(* LS Electric XG5000 project: LM1000_first_NC_program *)
(* PLC LSPLC *)
(* module base 0 slot 0: Input/Output Module:XMC-DN24 (DC 24V Input 8Points/TR output 16Points) *)
(* module base 0 slot 1: Internal Analog Input/Output:XMF-AH04E (A/D voltage/current 2 channels, D/A voltage 2 channels) *)
(* task Periodic Task: Kind=2 *)
(* task Initialization Task: Kind=1 *)
(* task NC Program: Kind=6 *)
VAR_GLOBAL
    NC_Ch1 : UINT := 1;
END_VAR

PROGRAM LDprogram (* task: Scan Program *)
VAR
    LS_CONNECT1 : LS_CONNECT;
    LS_DISCONNECT1 : LS_DISCONNECT;
    MC_HOMEALL1 : MC_HOMEALL;
    MC_POWERALL1 : MC_POWERALL;
    NC_CYCLESTART1 : NC_CYCLESTART;
    NC_LOADPROGRAM1 : NC_LOADPROGRAM;
    NC_RESET1 : NC_RESET;
    xConnect : BOOL;
    xHoming : BOOL;
    xLoadNCProgram : BOOL;
    xResetNCChannel : BOOL;
    xStartCycle : BOOL;
END_VAR
VAR_EXTERNAL
    NC_Ch1 : UINT;
END_VAR
VAR
    _e1 : F_TRIG;
END_VAR

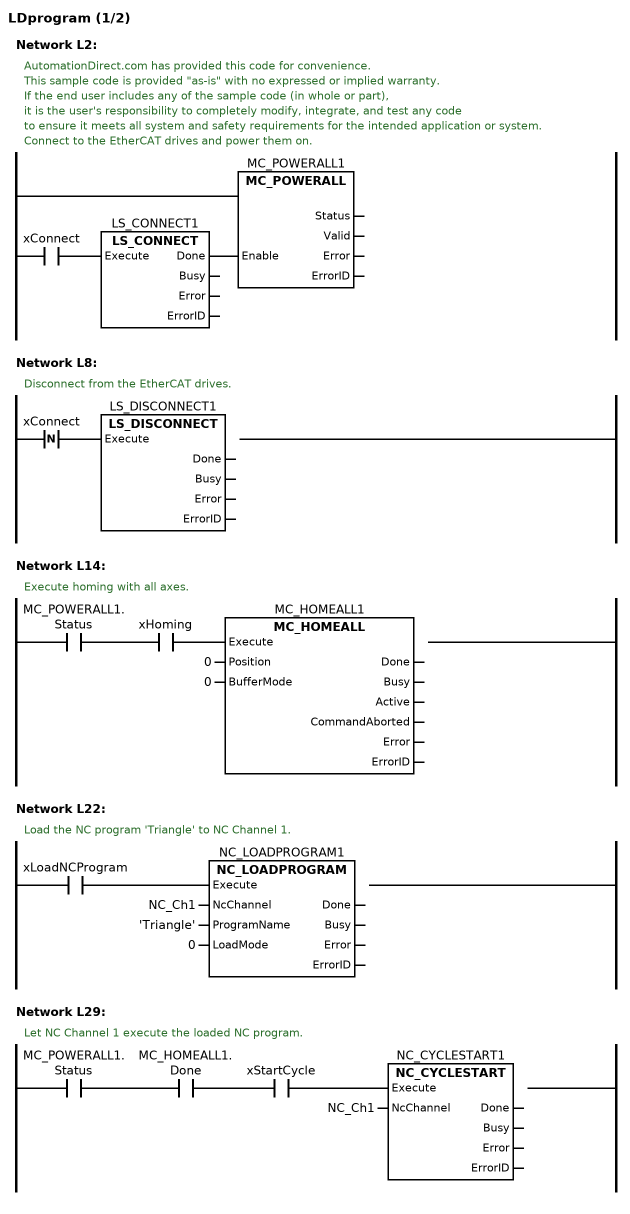
(* AutomationDirect.com has provided this code for convenience. / This sample code is provided "as-is" with no expressed or implied warranty. / If the end user includes any of the sample code (in whole or part), / it is the user's responsibility to completely modify, integrate, and test any code / to ensure it meets all system and safety requirements for the intended application or system. *)
(* Connect to the EtherCAT drives and power them on. *)
(* Rung L2 *)
LS_CONNECT1(Execute := xConnect);
MC_POWERALL1(Enable := LS_CONNECT1.Done);
(* Disconnect from the EtherCAT drives. *)
(* Rung L8 *)
_e1(CLK := xConnect);
LS_DISCONNECT1(Execute := _e1.Q);
(* Execute homing with all axes. *)
(* Rung L14 *)
MC_HOMEALL1(Execute := MC_POWERALL1.Status AND xHoming, Position := 0, BufferMode := 0);
(* Load the NC program 'Triangle' to NC Channel 1. *)
(* Rung L22 *)
NC_LOADPROGRAM1(Execute := xLoadNCProgram, NcChannel := NC_Ch1, ProgramName := 'Triangle', LoadMode := 0);
(* Let NC Channel 1 execute the loaded NC program. *)
(* Rung L29 *)
NC_CYCLESTART1(Execute := MC_POWERALL1.Status AND MC_HOMEALL1.Done AND xStartCycle, NcChannel := NC_Ch1);

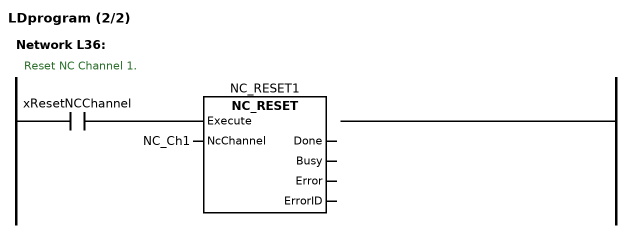
(* Reset NC Channel 1. *)
(* Rung L36 *)
NC_RESET1(Execute := xResetNCChannel, NcChannel := NC_Ch1);
END_PROGRAM

PROGRAM STprogram (* task: Scan Program *)
VAR
    F_TRIG1 : F_TRIG;
    LS_CONNECT1 : LS_CONNECT;
    LS_DISCONNECT1 : LS_DISCONNECT;
    MC_HOMEALL1 : MC_HOMEALL;
    MC_POWERALL1 : MC_POWERALL;
    NC_CYCLESTART1 : NC_CYCLESTART;
    NC_LOADPROGRAM1 : NC_LOADPROGRAM;
    NC_RESET1 : NC_RESET;
    xConnect : BOOL;
    xHoming : BOOL;
    xLoadNCProgram : BOOL;
    xRestNCChannel : BOOL;
    xStartCycle : BOOL;
END_VAR
VAR_EXTERNAL
    NC_Ch1 : UINT;
END_VAR
// AutomationDirect.com has provided this code for convenience. 
// This sample code is provided "as-is" with no expressed or implied warranty. 
// If the end user includes any of the sample code (in whole or part), 
// it is the user's responsibility to completely modify, integrate, and test any code 
// to ensure it meets all system and safety requirements for the intended application or system.


// Connect to the EtherCAT drives and power them on.
LS_CONNECT1(Execute:=xConnect, ErrorID=>LS_CONNECT1.ErrorID);
MC_POWERALL1(Enable:=LS_CONNECT1.Done, ErrorID=>MC_POWERALL1.ErrorID);

// Disconnect from the EtherCAT drives.
F_TRIG1(CLK:=xConnect);
LS_DISCONNECT1(Execute:=F_TRIG1.Q, ErrorID=>LS_DISCONNECT1.ErrorID);

// Execute homing with all axes.
MC_HOMEALL1(Execute:=(MC_POWERALL1.Status AND xHoming), Position:=0, BufferMode:=0, ErrorID=>MC_HOMEALL1.ErrorID);

// Load the NC program 'Triangle' to NC Channel 1.
NC_LOADPROGRAM1(Execute:=xLoadNCProgram, NcChannel:=NC_Ch1, ProgramName:='Triangle', LoadMode:=0, ErrorID=>NC_LOADPROGRAM1.ErrorID);

// Let NC Channel 1 execute the loaded NC program.
NC_CYCLESTART1(Execute:=(MC_POWERALL1.Status AND MC_HOMEALL1.Done AND xStartCycle), NcChannel:=NC_Ch1, ErrorID=>NC_CYCLESTART1.ErrorID);

// Reset NC Channel 1.
NC_RESET1(Execute:=xRestNCChannel, NcChannel:=NC_Ch1, ErrorID=>NC_RESET1.ErrorID);
END_PROGRAM

PROGRAM Triangle (* task: NC Program *)
% This is your first NC program.

G21 G90
G00 X100 Y100
G01 X300 Y100
G01 X200 Y200
G01 X100 Y100
M30
END_PROGRAM